{attribute 'qualified_only'}
TYPE SectionEnum :
(
	NULL_SECTION := 0,
	PAPER,
	CARDBOARD_CORNERGUARD,
	CHIPBOARD,
	WOOD_BUNK,
	OUTPUT,
	
	size
);
END_TYPE

(* stored: Version 1.1.0.1, ProductVersion 3.1.4024.11
   DUT SectionEnum: Id {ce069944-4100-460e-8745-53f394723540} *)
